PROGRAM MAIN
VAR
	a:INT;
	b:int;
END_VAR

a:=a+b;

END_PROGRAM

(* stored: Version 1.1.0.1, ProductVersion 3.1.4023.14
   POU MAIN: Id {2f0017be-33bf-42dd-a78a-5912f4f7a2cc}, SpecialFunc None *)
